Fanuc TP program (LS listing): mv_to_pick.ls

/PROG  MV_TO_PICK
/ATTR
DEFAULT_GROUP	= 1,*,*,*,*;
/MN
 : CALL MV_RETREAT ;
 :  ;
 : UFRAME_NUM=1 ;
 : UTOOL_NUM=1 ;
 : J PR[10:PICK_PERCH] 100% CNT100 ;
/POS
/END
